FUNCTION F_SAFETY_StatusFB_TO_OR : ST_SAFETY_FBOR
VAR_INPUT
	stFBStatus						: ST_SAFETY_FBStatus; 	(* Struktura ogolna *)
END_VAR

F_SAFETY_StatusFB_TO_OR.uStatus.stStatusWords 		:= stFBStatus;									(* Przepisanie *)
F_SAFETY_StatusFB_TO_OR.eState					 	:= stFBStatus.BState;							(* Ustawienie enum *)

END_FUNCTION

(* stored: Version 1.1.0.1, ProductVersion 3.1.4022.12
   POU F_SAFETY_StatusFB_TO_OR: Id {12d0749f-f096-40d1-a4d9-259f55ff4e49}, SpecialFunc None *)
